FUNCTION_BLOCK FB_2_VisionSkills EXTENDS FB_1_Skill
VAR_INPUT
	pOwnerCam: POINTER TO FB_1_Camera;
	CAM : REFERENCE TO FB_VN_GevCameraControl;
END_VAR
VAR_OUTPUT
END_VAR
VAR
	_Init_VisionSkill: BOOL;
END_VAR

pOwner := pOwnerCam;
IF pOwnerCam<>0 THEN
	CAM REF= pOwnerCam^.CAM;
END_IF

ACTION CYCLIC_VISIONSKILL:
IF NOT _Init_VisionSkill THEN
	_Init_VisionSkill:=TRUE;
	SETUP_VISIONSKILL();
END_IF


CYCLIC_SKILL();
END_ACTION

ACTION SETUP_VISIONSKILL:
pOwner := pOwnerCam;
IF pOwnerCam<>0 THEN
	CAM REF= pOwnerCam^.CAM;
END_IF
END_ACTION

END_FUNCTION_BLOCK

(* stored: Version 1.1.0.1, ProductVersion 3.1.4026.18
   POU FB_2_VisionSkills: Id {c094065f-2319-4570-a12a-5a88ea805ce7}, SpecialFunc None
   Action CYCLIC_VISIONSKILL: Id {a00d0d3e-61e2-40da-bba0-005e9199daed}
   Action SETUP_VISIONSKILL: Id {7da519fc-3c12-42b6-8bb9-d77a4915edef} *)
